TYPE ReadWrite_Enum :
(
	R_O := 0,
	R_W := 1
);
END_TYPE

(* stored: Version 1.1.0.1, ProductVersion 3.1.4024.11
   DUT ReadWrite_Enum: Id {1c690b1e-5ee8-45ac-87f8-f921bda423ab} *)
